// TIA Portal V21 export
DATA_BLOCK "db_TEST"   // DB1
{ S7_Optimized_Access := 'TRUE' }
// stored: InstanceOfName udt_TEST, InstanceOfType UDT
"udt_TEST"
   // VAR
   //    "a" : Bool;
   // END_VAR
BEGIN
END_DATA_BLOCK
